// TIA Portal V18 export
TYPE "UDT_SetPointsBasic"
// stored: IsFailsafeCompliant false
   STRUCT
      RATHeating : Array[1..3] of Real;   // C
      RATCooling : Array[1..3] of Real;   // C
      IAQ : Array[1..3] of Real;   // ppm
      BuildingdP : Array[1..3] of Real;   // Pa
   END_STRUCT;
   // RATHeating[1..2] := 20.0;
   // RATCooling[1..2] := 22.0;
   // IAQ[1..2] := 800.0;
   // BuildingdP[1..2] := 5.0;
END_TYPE
